PROGRAM main
VAR
	SW1 AT %IX0.3 : bool;
	SW2 AT %IX0.4 : bool;
	CR1 AT %QX2.0 : bool;
	CR2 AT %QX2.1 : bool;
	CR3 AT %QX0.0 : bool;
	CR : bool;
	CR4 : bool;
	CR5 : bool;
	CR6 : bool;
	CR7 : bool;
END_VAR

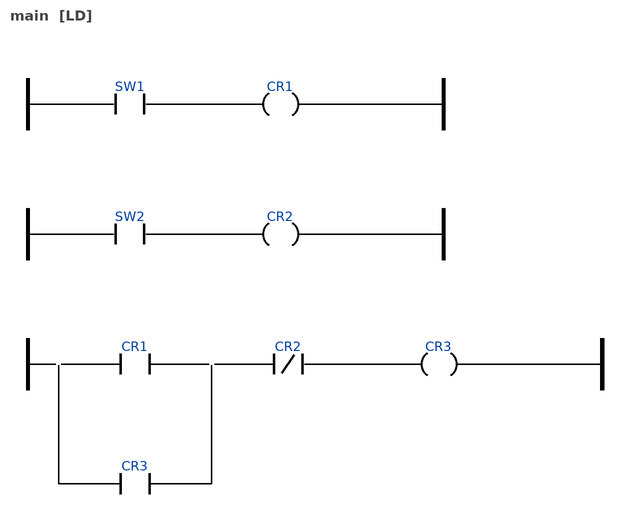
(* LD diagram, written out as Structured Text *)
CR1 := SW1;
CR2 := SW2;
CR3 := (CR1 OR CR3) AND NOT CR2;
END_PROGRAM
